# B&R Automation Studio project NAINV104C00R8L515F00 (part 15)

#### Act_OptP1081Navi.st
```iecst
ACTION Act_OptP1081Navi:

	IF tyP1081UsrMgmtUsrAccessRgt.tyNaviBack.tyBtnBack.bRtCompl = TRUE THEN
		tyP1081UsrMgmtUsrAccessRgt.tyNaviBack.tyBtnBack.bRtCompl	:= FALSE;
		tyP1081UsrMgmtUsrAccessRgt.tyNaviBack.tyBtnBack.bValue		:= FALSE;

		eChgPage	:= UIP1080UsrMgmt;
	END_IF

END_ACTION
```

#### Act_OptP1081Load.st
```iecst
ACTION Act_OptP1081Load:

	IF tyP1081UsrMgmtUsrAccessRgt.tyUsrAccessRgtSel.tyDrpDnLevel.bRtCompl = TRUE THEN
		tyP1081UsrMgmtUsrAccessRgt.tyUsrAccessRgtSel.tyDrpDnLevel.bRtCompl	:= FALSE;

		CASE tyP1081UsrMgmtUsrAccessRgt.tyUsrAccessRgtSel.tyDrpDnLevel.usiValueIdx OF
			0:
				p_tyP1081UsrMgmtUsrAccessRgt ACCESS ADR(tyP1081UsrMgmtUsrAccessRgt.tyUsrAccessRgtLvl1);
			1:
				p_tyP1081UsrMgmtUsrAccessRgt ACCESS ADR(tyP1081UsrMgmtUsrAccessRgt.tyUsrAccessRgtLvl2);
			2:
				p_tyP1081UsrMgmtUsrAccessRgt ACCESS ADR(tyP1081UsrMgmtUsrAccessRgt.tyUsrAccessRgtLvl3);
		END_CASE

	END_IF

END_ACTION
```

#### Act_OptP1081Save.st
```iecst
ACTION Act_OptP1081Save:

	//Level 1
	IF tyP1081UsrMgmtUsrAccessRgt.tyUsrAccessRgtLvl1.tyStringNm.bRtCompl 		OR tyP1081UsrMgmtUsrAccessRgt.tyUsrAccessRgtLvl1.tyBtnOps.bRtCompl
		OR tyP1081UsrMgmtUsrAccessRgt.tyUsrAccessRgtLvl1.tyBtnProdSel.bRtCompl	OR tyP1081UsrMgmtUsrAccessRgt.tyUsrAccessRgtLvl1.tyBtnMagSel.bRtCompl
		OR tyP1081UsrMgmtUsrAccessRgt.tyUsrAccessRgtLvl1.tyBtnMcInfo.bRtCompl	OR tyP1081UsrMgmtUsrAccessRgt.tyUsrAccessRgtLvl1.tyBtnAlm.bRtCompl
		OR tyP1081UsrMgmtUsrAccessRgt.tyUsrAccessRgtLvl1.tyBtnBffrInfo.bRtCompl	OR tyP1081UsrMgmtUsrAccessRgt.tyUsrAccessRgtLvl1.tyBtnOvenInfo.bRtCompl
		OR tyP1081UsrMgmtUsrAccessRgt.tyUsrAccessRgtLvl1.tyBtnMagInfo.bRtCompl	OR tyP1081UsrMgmtUsrAccessRgt.tyUsrAccessRgtLvl1.tyBtnLFCtrl.bRtCompl
		OR tyP1081UsrMgmtUsrAccessRgt.tyUsrAccessRgtLvl1.tyBtnManual.bRtCompl	OR tyP1081UsrMgmtUsrAccessRgt.tyUsrAccessRgtLvl1.tyBtnSimu.bRtCompl
		OR tyP1081UsrMgmtUsrAccessRgt.tyUsrAccessRgtLvl1.tyBtnProdSet.bRtCompl	OR tyP1081UsrMgmtUsrAccessRgt.tyUsrAccessRgtLvl1.tyBtnMagSet.bRtCompl
		OR tyP1081UsrMgmtUsrAccessRgt.tyUsrAccessRgtLvl1.tyBtnMcSet.bRtCompl	OR tyP1081UsrMgmtUsrAccessRgt.tyUsrAccessRgtLvl1.tyBtnLang.bRtCompl
		OR tyP1081UsrMgmtUsrAccessRgt.tyUsrAccessRgtLvl1.tyBtnLFSet.bRtCompl	OR tyP1081UsrMgmtUsrAccessRgt.tyUsrAccessRgtLvl1.tyBtnChgParam.bRtCompl
		OR tyP1081UsrMgmtUsrAccessRgt.tyUsrAccessRgtLvl1.tyBtnManualFBOnly.bRtCompl
		//Level 2
		OR tyP1081UsrMgmtUsrAccessRgt.tyUsrAccessRgtLvl2.tyStringNm.bRtCompl 	OR tyP1081UsrMgmtUsrAccessRgt.tyUsrAccessRgtLvl2.tyBtnOps.bRtCompl
		OR tyP1081UsrMgmtUsrAccessRgt.tyUsrAccessRgtLvl2.tyBtnProdSel.bRtCompl	OR tyP1081UsrMgmtUsrAccessRgt.tyUsrAccessRgtLvl2.tyBtnMagSel.bRtCompl
		OR tyP1081UsrMgmtUsrAccessRgt.tyUsrAccessRgtLvl2.tyBtnMcInfo.bRtCompl	OR tyP1081UsrMgmtUsrAccessRgt.tyUsrAccessRgtLvl2.tyBtnAlm.bRtCompl
		OR tyP1081UsrMgmtUsrAccessRgt.tyUsrAccessRgtLvl2.tyBtnBffrInfo.bRtCompl	OR tyP1081UsrMgmtUsrAccessRgt.tyUsrAccessRgtLvl2.tyBtnOvenInfo.bRtCompl
		OR tyP1081UsrMgmtUsrAccessRgt.tyUsrAccessRgtLvl2.tyBtnMagInfo.bRtCompl	OR tyP1081UsrMgmtUsrAccessRgt.tyUsrAccessRgtLvl2.tyBtnLFCtrl.bRtCompl
		OR tyP1081UsrMgmtUsrAccessRgt.tyUsrAccessRgtLvl2.tyBtnManual.bRtCompl	OR tyP1081UsrMgmtUsrAccessRgt.tyUsrAccessRgtLvl2.tyBtnSimu.bRtCompl
		OR tyP1081UsrMgmtUsrAccessRgt.tyUsrAccessRgtLvl2.tyBtnProdSet.bRtCompl	OR tyP1081UsrMgmtUsrAccessRgt.tyUsrAccessRgtLvl2.tyBtnMagSet.bRtCompl
		OR tyP1081UsrMgmtUsrAccessRgt.tyUsrAccessRgtLvl2.tyBtnMcSet.bRtCompl	OR tyP1081UsrMgmtUsrAccessRgt.tyUsrAccessRgtLvl2.tyBtnLang.bRtCompl
		OR tyP1081UsrMgmtUsrAccessRgt.tyUsrAccessRgtLvl2.tyBtnLFSet.bRtCompl	OR tyP1081UsrMgmtUsrAccessRgt.tyUsrAccessRgtLvl2.tyBtnChgParam.bRtCompl
		OR tyP1081UsrMgmtUsrAccessRgt.tyUsrAccessRgtLvl2.tyBtnManualFBOnly.bRtCompl

		//Level 3
		OR tyP1081UsrMgmtUsrAccessRgt.tyUsrAccessRgtLvl3.tyStringNm.bRtCompl 	OR tyP1081UsrMgmtUsrAccessRgt.tyUsrAccessRgtLvl3.tyBtnOps.bRtCompl
		OR tyP1081UsrMgmtUsrAccessRgt.tyUsrAccessRgtLvl3.tyBtnProdSel.bRtCompl	OR tyP1081UsrMgmtUsrAccessRgt.tyUsrAccessRgtLvl3.tyBtnMagSel.bRtCompl
		OR tyP1081UsrMgmtUsrAccessRgt.tyUsrAccessRgtLvl3.tyBtnMcInfo.bRtCompl	OR tyP1081UsrMgmtUsrAccessRgt.tyUsrAccessRgtLvl3.tyBtnAlm.bRtCompl
		OR tyP1081UsrMgmtUsrAccessRgt.tyUsrAccessRgtLvl3.tyBtnBffrInfo.bRtCompl	OR tyP1081UsrMgmtUsrAccessRgt.tyUsrAccessRgtLvl3.tyBtnOvenInfo.bRtCompl
		OR tyP1081UsrMgmtUsrAccessRgt.tyUsrAccessRgtLvl3.tyBtnMagInfo.bRtCompl	OR tyP1081UsrMgmtUsrAccessRgt.tyUsrAccessRgtLvl3.tyBtnLFCtrl.bRtCompl
		OR tyP1081UsrMgmtUsrAccessRgt.tyUsrAccessRgtLvl3.tyBtnManual.bRtCompl	OR tyP1081UsrMgmtUsrAccessRgt.tyUsrAccessRgtLvl3.tyBtnSimu.bRtCompl
		OR tyP1081UsrMgmtUsrAccessRgt.tyUsrAccessRgtLvl3.tyBtnProdSet.bRtCompl	OR tyP1081UsrMgmtUsrAccessRgt.tyUsrAccessRgtLvl3.tyBtnMagSet.bRtCompl
		OR tyP1081UsrMgmtUsrAccessRgt.tyUsrAccessRgtLvl3.tyBtnMcSet.bRtCompl	OR tyP1081UsrMgmtUsrAccessRgt.tyUsrAccessRgtLvl3.tyBtnLang.bRtCompl
		OR tyP1081UsrMgmtUsrAccessRgt.tyUsrAccessRgtLvl3.tyBtnLFSet.bRtCompl	OR tyP1081UsrMgmtUsrAccessRgt.tyUsrAccessRgtLvl3.tyBtnChgParam.bRtCompl
		OR tyP1081UsrMgmtUsrAccessRgt.tyUsrAccessRgtLvl3.tyBtnManualFBOnly.bRtCompl
		THEN

		fUIInRtStatHide(ADR(tyCommon.tySet.tyBtnSave.uiMaskRtStat));

		//Level 1
		tyP1081UsrMgmtUsrAccessRgt.tyUsrAccessRgtLvl1.tyStringNm.bRtCompl 		:= FALSE;
		tyP1081UsrMgmtUsrAccessRgt.tyUsrAccessRgtLvl1.tyBtnOps.bRtCompl 		:= FALSE;
		tyP1081UsrMgmtUsrAccessRgt.tyUsrAccessRgtLvl1.tyBtnProdSel.bRtCompl 	:= FALSE;
		tyP1081UsrMgmtUsrAccessRgt.tyUsrAccessRgtLvl1.tyBtnMagSel.bRtCompl 		:= FALSE;
		tyP1081UsrMgmtUsrAccessRgt.tyUsrAccessRgtLvl1.tyBtnMcInfo.bRtCompl		:= FALSE;
		tyP1081UsrMgmtUsrAccessRgt.tyUsrAccessRgtLvl1.tyBtnAlm.bRtCompl			:= FALSE;
		tyP1081UsrMgmtUsrAccessRgt.tyUsrAccessRgtLvl1.tyBtnBffrInfo.bRtCompl	:= FALSE;
		tyP1081UsrMgmtUsrAccessRgt.tyUsrAccessRgtLvl1.tyBtnOvenInfo.bRtCompl	:= FALSE;
		tyP1081UsrMgmtUsrAccessRgt.tyUsrAccessRgtLvl1.tyBtnMagInfo.bRtCompl		:= FALSE;
		tyP1081UsrMgmtUsrAccessRgt.tyUsrAccessRgtLvl1.tyBtnLFCtrl.bRtCompl		:= FALSE;
		tyP1081UsrMgmtUsrAccessRgt.tyUsrAccessRgtLvl1.tyBtnManual.bRtCompl		:= FALSE;
		tyP1081UsrMgmtUsrAccessRgt.tyUsrAccessRgtLvl1.tyBtnSimu.bRtCompl		:= FALSE;
		tyP1081UsrMgmtUsrAccessRgt.tyUsrAccessRgtLvl1.tyBtnProdSet.bRtCompl		:= FALSE;
		tyP1081UsrMgmtUsrAccessRgt.tyUsrAccessRgtLvl1.tyBtnMagSet.bRtCompl		:= FALSE;
		tyP1081UsrMgmtUsrAccessRgt.tyUsrAccessRgtLvl1.tyBtnMcSet.bRtCompl		:= FALSE;
		tyP1081UsrMgmtUsrAccessRgt.tyUsrAccessRgtLvl1.tyBtnLang.bRtCompl		:= FALSE;
		tyP1081UsrMgmtUsrAccessRgt.tyUsrAccessRgtLvl1.tyBtnLFSet.bRtCompl		:= FALSE;
		tyP1081UsrMgmtUsrAccessRgt.tyUsrAccessRgtLvl1.tyBtnChgParam.bRtCompl	:= FALSE;
		tyP1081UsrMgmtUsrAccessRgt.tyUsrAccessRgtLvl1.tyBtnManualFBOnly.bRtCompl:= FALSE;

		//Level 2
		tyP1081UsrMgmtUsrAccessRgt.tyUsrAccessRgtLvl2.tyStringNm.bRtCompl 		:= FALSE;
		tyP1081UsrMgmtUsrAccessRgt.tyUsrAccessRgtLvl2.tyBtnOps.bRtCompl 		:= FALSE;
		tyP1081UsrMgmtUsrAccessRgt.tyUsrAccessRgtLvl2.tyBtnProdSel.bRtCompl 	:= FALSE;
		tyP1081UsrMgmtUsrAccessRgt.tyUsrAccessRgtLvl2.tyBtnMagSel.bRtCompl 		:= FALSE;
		tyP1081UsrMgmtUsrAccessRgt.tyUsrAccessRgtLvl2.tyBtnMcInfo.bRtCompl		:= FALSE;
		tyP1081UsrMgmtUsrAccessRgt.tyUsrAccessRgtLvl2.tyBtnAlm.bRtCompl			:= FALSE;
		tyP1081UsrMgmtUsrAccessRgt.tyUsrAccessRgtLvl2.tyBtnBffrInfo.bRtCompl	:= FALSE;
		tyP1081UsrMgmtUsrAccessRgt.tyUsrAccessRgtLvl2.tyBtnOvenInfo.bRtCompl	:= FALSE;
		tyP1081UsrMgmtUsrAccessRgt.tyUsrAccessRgtLvl2.tyBtnMagInfo.bRtCompl		:= FALSE;
		tyP1081UsrMgmtUsrAccessRgt.tyUsrAccessRgtLvl2.tyBtnLFCtrl.bRtCompl		:= FALSE;
		tyP1081UsrMgmtUsrAccessRgt.tyUsrAccessRgtLvl2.tyBtnManual.bRtCompl		:= FALSE;
		tyP1081UsrMgmtUsrAccessRgt.tyUsrAccessRgtLvl2.tyBtnSimu.bRtCompl		:= FALSE;
		tyP1081UsrMgmtUsrAccessRgt.tyUsrAccessRgtLvl2.tyBtnProdSet.bRtCompl		:= FALSE;
		tyP1081UsrMgmtUsrAccessRgt.tyUsrAccessRgtLvl2.tyBtnMagSet.bRtCompl		:= FALSE;
		tyP1081UsrMgmtUsrAccessRgt.tyUsrAccessRgtLvl2.tyBtnMcSet.bRtCompl		:= FALSE;
		tyP1081UsrMgmtUsrAccessRgt.tyUsrAccessRgtLvl2.tyBtnLang.bRtCompl		:= FALSE;
		tyP1081UsrMgmtUsrAccessRgt.tyUsrAccessRgtLvl2.tyBtnLFSet.bRtCompl		:= FALSE;
		tyP1081UsrMgmtUsrAccessRgt.tyUsrAccessRgtLvl2.tyBtnChgParam.bRtCompl	:= FALSE;
		tyP1081UsrMgmtUsrAccessRgt.tyUsrAccessRgtLvl2.tyBtnManualFBOnly.bRtCompl:= FALSE;

		//Level 3
		tyP1081UsrMgmtUsrAccessRgt.tyUsrAccessRgtLvl3.tyStringNm.bRtCompl 		:= FALSE;
		tyP1081UsrMgmtUsrAccessRgt.tyUsrAccessRgtLvl3.tyBtnOps.bRtCompl 		:= FALSE;
		tyP1081UsrMgmtUsrAccessRgt.tyUsrAccessRgtLvl3.tyBtnProdSel.bRtCompl 	:= FALSE;
		tyP1081UsrMgmtUsrAccessRgt.tyUsrAccessRgtLvl3.tyBtnMagSel.bRtCompl 		:= FALSE;
		tyP1081UsrMgmtUsrAccessRgt.tyUsrAccessRgtLvl3.tyBtnMcInfo.bRtCompl		:= FALSE;
		tyP1081UsrMgmtUsrAccessRgt.tyUsrAccessRgtLvl3.tyBtnAlm.bRtCompl			:= FALSE;
		tyP1081UsrMgmtUsrAccessRgt.tyUsrAccessRgtLvl3.tyBtnBffrInfo.bRtCompl	:= FALSE;
		tyP1081UsrMgmtUsrAccessRgt.tyUsrAccessRgtLvl3.tyBtnOvenInfo.bRtCompl	:= FALSE;
		tyP1081UsrMgmtUsrAccessRgt.tyUsrAccessRgtLvl3.tyBtnMagInfo.bRtCompl		:= FALSE;
		tyP1081UsrMgmtUsrAccessRgt.tyUsrAccessRgtLvl3.tyBtnLFCtrl.bRtCompl		:= FALSE;
		tyP1081UsrMgmtUsrAccessRgt.tyUsrAccessRgtLvl3.tyBtnManual.bRtCompl		:= FALSE;
		tyP1081UsrMgmtUsrAccessRgt.tyUsrAccessRgtLvl3.tyBtnSimu.bRtCompl		:= FALSE;
		tyP1081UsrMgmtUsrAccessRgt.tyUsrAccessRgtLvl3.tyBtnProdSet.bRtCompl		:= FALSE;
		tyP1081UsrMgmtUsrAccessRgt.tyUsrAccessRgtLvl3.tyBtnMagSet.bRtCompl		:= FALSE;
		tyP1081UsrMgmtUsrAccessRgt.tyUsrAccessRgtLvl3.tyBtnMcSet.bRtCompl		:= FALSE;
		tyP1081UsrMgmtUsrAccessRgt.tyUsrAccessRgtLvl3.tyBtnLang.bRtCompl		:= FALSE;
		tyP1081UsrMgmtUsrAccessRgt.tyUsrAccessRgtLvl3.tyBtnLFSet.bRtCompl		:= FALSE;
		tyP1081UsrMgmtUsrAccessRgt.tyUsrAccessRgtLvl3.tyBtnChgParam.bRtCompl	:= FALSE;
		tyP1081UsrMgmtUsrAccessRgt.tyUsrAccessRgtLvl3.tyBtnManualFBOnly.bRtCompl:= FALSE;

	END_IF

	IF tyCommon.tySet.tyBtnSave.bRtCompl = TRUE THEN
		//Save Param
		CASE tyP1081UsrMgmtUsrAccessRgt.tyUsrAccessRgtSel.tyDrpDnLevel.usiValueIdx OF
			0:
				tyUsrMgmtAccessRightLvl1Wr.sNm			:= tyP1081UsrMgmtUsrAccessRgt.tyUsrAccessRgtLvl1.tyStringNm.sValue;
				tyUsrMgmtAccessRightLvl1Wr.bOpt			:= tyP1081UsrMgmtUsrAccessRgt.tyUsrAccessRgtLvl1.tyBtnOps.bValue;
				tyUsrMgmtAccessRightLvl1Wr.bProdSel		:= tyP1081UsrMgmtUsrAccessRgt.tyUsrAccessRgtLvl1.tyBtnProdSel.bValue;
				tyUsrMgmtAccessRightLvl1Wr.bMagSel		:= tyP1081UsrMgmtUsrAccessRgt.tyUsrAccessRgtLvl1.tyBtnMagSel.bValue;
				tyUsrMgmtAccessRightLvl1Wr.bMcInfo		:= tyP1081UsrMgmtUsrAccessRgt.tyUsrAccessRgtLvl1.tyBtnMcInfo.bValue;
				tyUsrMgmtAccessRightLvl1Wr.bAlm			:= tyP1081UsrMgmtUsrAccessRgt.tyUsrAccessRgtLvl1.tyBtnAlm.bValue;
				tyUsrMgmtAccessRightLvl1Wr.bBffrInfo	:= tyP1081UsrMgmtUsrAccessRgt.tyUsrAccessRgtLvl1.tyBtnBffrInfo.bValue;
				tyUsrMgmtAccessRightLvl1Wr.bOvenInfo	:= tyP1081UsrMgmtUsrAccessRgt.tyUsrAccessRgtLvl1.tyBtnOvenInfo.bValue;
				tyUsrMgmtAccessRightLvl1Wr.bMagInfo		:= tyP1081UsrMgmtUsrAccessRgt.tyUsrAccessRgtLvl1.tyBtnMagInfo.bValue;
				tyUsrMgmtAccessRightLvl1Wr.bLFCtrl		:= tyP1081UsrMgmtUsrAccessRgt.tyUsrAccessRgtLvl1.tyBtnLFCtrl.bValue;
				tyUsrMgmtAccessRightLvl1Wr.bManual		:= tyP1081UsrMgmtUsrAccessRgt.tyUsrAccessRgtLvl1.tyBtnManual.bValue;
				tyUsrMgmtAccessRightLvl1Wr.bSimulation	:= tyP1081UsrMgmtUsrAccessRgt.tyUsrAccessRgtLvl1.tyBtnSimu.bValue;
				tyUsrMgmtAccessRightLvl1Wr.bProdSet		:= tyP1081UsrMgmtUsrAccessRgt.tyUsrAccessRgtLvl1.tyBtnProdSet.bValue;
				tyUsrMgmtAccessRightLvl1Wr.bMagSet		:= tyP1081UsrMgmtUsrAccessRgt.tyUsrAccessRgtLvl1.tyBtnMagSet.bValue;
				tyUsrMgmtAccessRightLvl1Wr.bMcSet		:= tyP1081UsrMgmtUsrAccessRgt.tyUsrAccessRgtLvl1.tyBtnMcSet.bValue;
				tyUsrMgmtAccessRightLvl1Wr.bLang		:= tyP1081UsrMgmtUsrAccessRgt.tyUsrAccessRgtLvl1.tyBtnLang.bValue;
				tyUsrMgmtAccessRightLvl1Wr.bLFSet		:= tyP1081UsrMgmtUsrAccessRgt.tyUsrAccessRgtLvl1.tyBtnLFSet.bValue;
				tyUsrMgmtAccessRightLvl1Wr.bChgParam	:= tyP1081UsrMgmtUsrAccessRgt.tyUsrAccessRgtLvl1.tyBtnChgParam.bValue;
				tyUsrMgmtAccessRightLvl1Wr.bManualFBOnly:= tyP1081UsrMgmtUsrAccessRgt.tyUsrAccessRgtLvl1.tyBtnManualFBOnly.bValue;

			1:
				tyUsrMgmtAccessRightLvl2Wr.sNm			:= tyP1081UsrMgmtUsrAccessRgt.tyUsrAccessRgtLvl2.tyStringNm.sValue;
				tyUsrMgmtAccessRightLvl2Wr.bOpt			:= tyP1081UsrMgmtUsrAccessRgt.tyUsrAccessRgtLvl2.tyBtnOps.bValue;
				tyUsrMgmtAccessRightLvl2Wr.bProdSel		:= tyP1081UsrMgmtUsrAccessRgt.tyUsrAccessRgtLvl2.tyBtnProdSel.bValue;
				tyUsrMgmtAccessRightLvl2Wr.bMagSel		:= tyP1081UsrMgmtUsrAccessRgt.tyUsrAccessRgtLvl2.tyBtnMagSel.bValue;
				tyUsrMgmtAccessRightLvl2Wr.bMcInfo		:= tyP1081UsrMgmtUsrAccessRgt.tyUsrAccessRgtLvl2.tyBtnMcInfo.bValue;
				tyUsrMgmtAccessRightLvl2Wr.bAlm			:= tyP1081UsrMgmtUsrAccessRgt.tyUsrAccessRgtLvl2.tyBtnAlm.bValue;
				tyUsrMgmtAccessRightLvl2Wr.bBffrInfo	:= tyP1081UsrMgmtUsrAccessRgt.tyUsrAccessRgtLvl2.tyBtnBffrInfo.bValue;
				tyUsrMgmtAccessRightLvl2Wr.bOvenInfo	:= tyP1081UsrMgmtUsrAccessRgt.tyUsrAccessRgtLvl2.tyBtnOvenInfo.bValue;
				tyUsrMgmtAccessRightLvl2Wr.bMagInfo		:= tyP1081UsrMgmtUsrAccessRgt.tyUsrAccessRgtLvl2.tyBtnMagInfo.bValue;
				tyUsrMgmtAccessRightLvl2Wr.bLFCtrl		:= tyP1081UsrMgmtUsrAccessRgt.tyUsrAccessRgtLvl2.tyBtnLFCtrl.bValue;
				tyUsrMgmtAccessRightLvl2Wr.bManual		:= tyP1081UsrMgmtUsrAccessRgt.tyUsrAccessRgtLvl2.tyBtnManual.bValue;
				tyUsrMgmtAccessRightLvl2Wr.bSimulation	:= tyP1081UsrMgmtUsrAccessRgt.tyUsrAccessRgtLvl2.tyBtnSimu.bValue;
				tyUsrMgmtAccessRightLvl2Wr.bProdSet		:= tyP1081UsrMgmtUsrAccessRgt.tyUsrAccessRgtLvl2.tyBtnProdSet.bValue;
				tyUsrMgmtAccessRightLvl2Wr.bMagSet		:= tyP1081UsrMgmtUsrAccessRgt.tyUsrAccessRgtLvl2.tyBtnMagSet.bValue;
				tyUsrMgmtAccessRightLvl2Wr.bMcSet		:= tyP1081UsrMgmtUsrAccessRgt.tyUsrAccessRgtLvl2.tyBtnMcSet.bValue;
				tyUsrMgmtAccessRightLvl2Wr.bLang		:= tyP1081UsrMgmtUsrAccessRgt.tyUsrAccessRgtLvl2.tyBtnLang.bValue;
				tyUsrMgmtAccessRightLvl2Wr.bLFSet		:= tyP1081UsrMgmtUsrAccessRgt.tyUsrAccessRgtLvl2.tyBtnLFSet.bValue;
				tyUsrMgmtAccessRightLvl2Wr.bChgParam	:= tyP1081UsrMgmtUsrAccessRgt.tyUsrAccessRgtLvl2.tyBtnChgParam.bValue;
				tyUsrMgmtAccessRightLvl2Wr.bManualFBOnly:= tyP1081UsrMgmtUsrAccessRgt.tyUsrAccessRgtLvl2.tyBtnManualFBOnly.bValue;

			2:
				tyUsrMgmtAccessRightLvl3Wr.sNm			:= tyP1081UsrMgmtUsrAccessRgt.tyUsrAccessRgtLvl3.tyStringNm.sValue;
				tyUsrMgmtAccessRightLvl3Wr.bOpt			:= tyP1081UsrMgmtUsrAccessRgt.tyUsrAccessRgtLvl3.tyBtnOps.bValue;
				tyUsrMgmtAccessRightLvl3Wr.bProdSel		:= tyP1081UsrMgmtUsrAccessRgt.tyUsrAccessRgtLvl3.tyBtnProdSel.bValue;
				tyUsrMgmtAccessRightLvl3Wr.bMagSel		:= tyP1081UsrMgmtUsrAccessRgt.tyUsrAccessRgtLvl3.tyBtnMagSel.bValue;
				tyUsrMgmtAccessRightLvl3Wr.bMcInfo		:= tyP1081UsrMgmtUsrAccessRgt.tyUsrAccessRgtLvl3.tyBtnMcInfo.bValue;
				tyUsrMgmtAccessRightLvl3Wr.bAlm			:= tyP1081UsrMgmtUsrAccessRgt.tyUsrAccessRgtLvl3.tyBtnAlm.bValue;
				tyUsrMgmtAccessRightLvl3Wr.bBffrInfo	:= tyP1081UsrMgmtUsrAccessRgt.tyUsrAccessRgtLvl3.tyBtnBffrInfo.bValue;
				tyUsrMgmtAccessRightLvl3Wr.bOvenInfo	:= tyP1081UsrMgmtUsrAccessRgt.tyUsrAccessRgtLvl3.tyBtnOvenInfo.bValue;
				tyUsrMgmtAccessRightLvl3Wr.bMagInfo		:= tyP1081UsrMgmtUsrAccessRgt.tyUsrAccessRgtLvl3.tyBtnMagInfo.bValue;
				tyUsrMgmtAccessRightLvl3Wr.bLFCtrl		:= tyP1081UsrMgmtUsrAccessRgt.tyUsrAccessRgtLvl3.tyBtnLFCtrl.bValue;
				tyUsrMgmtAccessRightLvl3Wr.bManual		:= tyP1081UsrMgmtUsrAccessRgt.tyUsrAccessRgtLvl3.tyBtnManual.bValue;
				tyUsrMgmtAccessRightLvl3Wr.bSimulation	:= tyP1081UsrMgmtUsrAccessRgt.tyUsrAccessRgtLvl3.tyBtnSimu.bValue;
				tyUsrMgmtAccessRightLvl3Wr.bProdSet		:= tyP1081UsrMgmtUsrAccessRgt.tyUsrAccessRgtLvl3.tyBtnProdSet.bValue;
				tyUsrMgmtAccessRightLvl3Wr.bMagSet		:= tyP1081UsrMgmtUsrAccessRgt.tyUsrAccessRgtLvl3.tyBtnMagSet.bValue;
				tyUsrMgmtAccessRightLvl3Wr.bMcSet		:= tyP1081UsrMgmtUsrAccessRgt.tyUsrAccessRgtLvl3.tyBtnMcSet.bValue;
				tyUsrMgmtAccessRightLvl3Wr.bLang		:= tyP1081UsrMgmtUsrAccessRgt.tyUsrAccessRgtLvl3.tyBtnLang.bValue;
				tyUsrMgmtAccessRightLvl3Wr.bLFSet		:= tyP1081UsrMgmtUsrAccessRgt.tyUsrAccessRgtLvl3.tyBtnLFSet.bValue;
				tyUsrMgmtAccessRightLvl3Wr.bChgParam	:= tyP1081UsrMgmtUsrAccessRgt.tyUsrAccessRgtLvl3.tyBtnChgParam.bValue;
				tyUsrMgmtAccessRightLvl3Wr.bManualFBOnly:= tyP1081UsrMgmtUsrAccessRgt.tyUsrAccessRgtLvl3.tyBtnManualFBOnly.bValue;

		END_CASE

		eUsrMgmtAct	:= UsrMgmtActSaveAccessRight;

		IF p_eUsrMgmtStat = UsrMgmtActSaveAccessRight AND p_eUsrMgmtStatus = Done THEN
			eUsrMgmtAct	:= UsrMgmtActIdle;

			//Backup Param
			tyP1081UsrMgmtUsrAccessRgt.tyUsrAccessRgtLvl1BkUp	:= tyP1081UsrMgmtUsrAccessRgt.tyUsrAccessRgtLvl1;
			tyP1081UsrMgmtUsrAccessRgt.tyUsrAccessRgtLvl2BkUp	:= tyP1081UsrMgmtUsrAccessRgt.tyUsrAccessRgtLvl2;
			tyP1081UsrMgmtUsrAccessRgt.tyUsrAccessRgtLvl3BkUp	:= tyP1081UsrMgmtUsrAccessRgt.tyUsrAccessRgtLvl3;

			CASE tyP1081UsrMgmtUsrAccessRgt.tyUsrAccessRgtSel.tyDrpDnLevel.usiValueIdx OF
				0:
					tyProperty.tyUITxtSnippets.sUsrMgmtUsrLv1Nm	:= tyP1081UsrMgmtUsrAccessRgt.tyUsrAccessRgtLvl1.tyStringNm.sValue;
				1:
					tyProperty.tyUITxtSnippets.sUsrMgmtUsrLv2Nm	:= tyP1081UsrMgmtUsrAccessRgt.tyUsrAccessRgtLvl2.tyStringNm.sValue;
				2:
					tyProperty.tyUITxtSnippets.sUsrMgmtUsrLv3Nm	:= tyP1081UsrMgmtUsrAccessRgt.tyUsrAccessRgtLvl3.tyStringNm.sValue;
			END_CASE

			tyCommon.tySet.tyBtnSave.bRtCompl	:= FALSE;

			fUIInRtStatOff(ADR(tyCommon.tySet.tyBtnSave.uiMaskRtStat));

		ELSIF p_eUsrMgmtStatus = Error THEN
			p_tyC0008MsgBox ACCESS ADR(tyP1081UsrMgmtUsrAccessRgt.tyMsgBoxSaveErr);

			IF tyP1081UsrMgmtUsrAccessRgt.tyMsgBoxSaveErr.tyBtnNo.bRtCompl = TRUE THEN
				tyP1081UsrMgmtUsrAccessRgt.tyMsgBoxSaveErr.tyBtnNo.bRtCompl	:= FALSE;
				tyP1081UsrMgmtUsrAccessRgt.tyMsgBoxSaveErr.tyBtnNo.bValue	:= FALSE;

				p_tyC0008MsgBox ACCESS ADR(tyP1081UsrMgmtUsrAccessRgt.tyMsgBoxHide);

				//Recover Param
				tyUsrMgmtAccessRightLvl1Wr	:= p_tyUsrMgmtFullData.tyAccessRightLvl1;
				tyUsrMgmtAccessRightLvl2Wr	:= p_tyUsrMgmtFullData.tyAccessRightLvl2;
				tyUsrMgmtAccessRightLvl3Wr	:= p_tyUsrMgmtFullData.tyAccessRightLvl3;

				tyP1081UsrMgmtUsrAccessRgt.tyUsrAccessRgtLvl1	:= tyP1081UsrMgmtUsrAccessRgt.tyUsrAccessRgtLvl1BkUp;
				tyP1081UsrMgmtUsrAccessRgt.tyUsrAccessRgtLvl2	:= tyP1081UsrMgmtUsrAccessRgt.tyUsrAccessRgtLvl2BkUp;
				tyP1081UsrMgmtUsrAccessRgt.tyUsrAccessRgtLvl3	:= tyP1081UsrMgmtUsrAccessRgt.tyUsrAccessRgtLvl3BkUp;

				tyCommon.tySet.tyBtnSave.bRtCompl	:= FALSE;

				fUIInRtStatOff(ADR(tyCommon.tySet.tyBtnSave.uiMaskRtStat));

			END_IF

		END_IF

	END_IF

END_ACTION
```

#### Act_OptP1081Keypad.st
```iecst
ACTION Act_OptP1081Keypad:

	IF fUIOutRtStatTPIsOpen(ADR(tyP1081UsrMgmtUsrAccessRgt.tyUsrAccessRgtLvl1.tyStringNm.uiRtStat)) = TRUE THEN
		tyProperty.tyKeypad.tyTxtTitle.sTxt	:= tyP1081UsrMgmtUsrAccessRgt.tyUsrAccessRgtLvl1.tyStringNm.sKeypadTitle;

	ELSIF fUIOutRtStatTPIsOpen(ADR(tyP1081UsrMgmtUsrAccessRgt.tyUsrAccessRgtLvl2.tyStringNm.uiRtStat)) = TRUE THEN
		tyProperty.tyKeypad.tyTxtTitle.sTxt	:= tyP1081UsrMgmtUsrAccessRgt.tyUsrAccessRgtLvl2.tyStringNm.sKeypadTitle;

	ELSIF fUIOutRtStatTPIsOpen(ADR(tyP1081UsrMgmtUsrAccessRgt.tyUsrAccessRgtLvl3.tyStringNm.uiRtStat)) = TRUE THEN
		tyProperty.tyKeypad.tyTxtTitle.sTxt	:= tyP1081UsrMgmtUsrAccessRgt.tyUsrAccessRgtLvl3.tyStringNm.sKeypadTitle;

	END_IF

END_ACTION
```

#### Act_OptP0002ToP1081UnlockCoverPB.st
```iecst
ACTION Act_OptP0002ToP1081UnlockCoverPB:

	IF p_tyNtParamCurr.tyDOSettings.diBypassTopCover1 > 0 THEN

		IF p_bAlarmErr THEN
			bCoverPB1Timer := FALSE;
			fbCoverPB1CountDownTm( IN := FALSE);
			tyP0200OpsGen.tyOps.tyBtnBypassTopCover1.bValue 	:=FALSE;
			tyP0201OpsConv.tyOps.tyBtnBypassTopCover1.bValue	:=FALSE;
		END_IF

		//Physical Unlock Cover Button 1
		IF EDGENEG(p_tyDI.bCoverUnlockPB1) THEN
			IF p_tyDI.bCoverSWSig2 = TRUE THEN
				IF tyP0200OpsGen.tyOps.tyBtnBypassTopCover1.bValue = FALSE THEN
					tyP0200OpsGen.tyOps.tyBtnBypassTopCover1.bValue 	:= TRUE;
					tyP0201OpsConv.tyOps.tyBtnBypassTopCover1.bValue	:= tyP0200OpsGen.tyOps.tyBtnBypassTopCover1.bValue;
					bCoverPB1Timer := TRUE;
				ELSE
					tyP0200OpsGen.tyOps.tyBtnBypassTopCover1.bValue 	:= FALSE;
					tyP0201OpsConv.tyOps.tyBtnBypassTopCover1.bValue	:= tyP0200OpsGen.tyOps.tyBtnBypassTopCover1.bValue;
					bCoverPB1Timer := FALSE;
				END_IF
			END_IF
		END_IF

		//Control
		IF tyP0200OpsGen.tyOps.tyBtnBypassTopCover1.bRtCompl = TRUE THEN //ok
			tyP0200OpsGen.tyOps.tyBtnBypassTopCover1.bRtCompl	:= FALSE;
			IF p_tyDI.bCoverSWSig2 = TRUE THEN
				tyP0201OpsConv.tyOps.tyBtnBypassTopCover1.bValue	:= tyP0200OpsGen.tyOps.tyBtnBypassTopCover1.bValue;
				IF tyP0200OpsGen.tyOps.tyBtnBypassTopCover1.bValue = TRUE THEN
					bCoverPB1Timer := TRUE;
				ELSE
					bCoverPB1Timer := FALSE;
				END_IF
			ELSE
				tyP0200OpsGen.tyOps.tyBtnBypassTopCover1.bValue 	:= TRUE;
				tyP0201OpsConv.tyOps.tyBtnBypassTopCover1.bValue	:= tyP0200OpsGen.tyOps.tyBtnBypassTopCover1.bValue;
			END_IF

		ELSIF tyP0201OpsConv.tyOps.tyBtnBypassTopCover1.bRtCompl = TRUE THEN //ok
			tyP0201OpsConv.tyOps.tyBtnBypassTopCover1.bRtCompl	:= FALSE;
			IF p_tyDI.bCoverSWSig = TRUE THEN
				tyP0200OpsGen.tyOps.tyBtnBypassTopCover1.bValue	:= tyP0201OpsConv.tyOps.tyBtnBypassTopCover1.bValue;
				IF tyP0201OpsConv.tyOps.tyBtnBypassTopCover1.bValue = TRUE THEN
					bCoverPB1Timer := TRUE;
				ELSE
					bCoverPB1Timer := FALSE;
				END_IF
			ELSE
				tyP0201OpsConv.tyOps.tyBtnBypassTopCover1.bValue 	:= TRUE;
				tyP0200OpsGen.tyOps.tyBtnBypassTopCover1.bValue		:= tyP0201OpsConv.tyOps.tyBtnBypassTopCover1.bValue;
			END_IF

		END_IF

		bBypassTopCover1	:= ( tyP0200OpsGen.tyOps.tyBtnBypassTopCover1.bValue) OR ( tyP0201OpsConv.tyOps.tyBtnBypassTopCover1.bValue);

		//Condition Allow
		IF (tyP0201OpsConv.tyOps.tyBtnBypassTopCover1.bValue = TRUE) THEN

			IF p_tyNtParamCurr.tyDISettings.diSafetySigFromUS > 0 THEN
				bUnlockCover1Req	:= TRUE;

				IF (p_bOpsInvertStepAWMove = FALSE) AND (p_eConvStatus <> Busy AND p_eInvertStatus <> Busy )AND
					(( p_tyDI.bInShutterCloseRS AND p_tyDI.bOutShutterCloseRS AND p_bOpsSafeMode) OR p_bOpsRun=FALSE) AND (p_tyDI.bSafetySigFromUS AND p_tyDI.bSafetySigFromDS )  THEN

					bTopCoverSwitchCoil1	:= FALSE;
				ELSE
					bTopCoverSwitchCoil1	:= TRUE;
				END_IF

			ELSE
				IF (p_bOpsInvertStepAWMove = FALSE) AND (p_eConvStatus <> Busy AND p_eInvertStatus <> Busy )AND
					((p_tyDI.bInShutterCloseRS AND p_tyDI.bOutShutterCloseRS AND p_bOpsSafeMode) OR p_bOpsRun=FALSE) THEN

					bTopCoverSwitchCoil1	:= FALSE;
				ELSE
					bTopCoverSwitchCoil1	:= TRUE;
				END_IF

			END_IF

		ELSE
			bTopCoverSwitchCoil1	:= TRUE;
			IF p_tyNtParamCurr.tyDISettings.diSafetySigFromUS > 0 THEN
				bUnlockCover1Req	:= FALSE;
				//bTopCvrUnlckToDS	:= FALSE;
			END_IF

		END_IF

		//Button Appearance
		IF bCoverPBLED1 THEN //bTopCoverSwitchCoil1 = FALSE AND tyP0200OpsGen.tyOps.tyBtnBypassTopCover1.bValue = TRUE THEN
			tyP0201OpsConv.tyOps.tyBitmapBypassTopCover1.usiValueIdx	:= 0;
			tyP0200OpsGen.tyOps.tyBitmapBypassTopCover1.usiValueIdx		:= 0;
		ELSE
			tyP0201OpsConv.tyOps.tyBitmapBypassTopCover1.usiValueIdx	:= 2;
			tyP0200OpsGen.tyOps.tyBitmapBypassTopCover1.usiValueIdx		:= 2;
		END_IF

	END_IF

	//lED 1&2

	// LED 1 & 2
	IF bTopCoverSwitchCoil1 = FALSE AND tyP0200OpsGen.tyOps.tyBtnBypassTopCover1.bValue = TRUE THEN
		bCoverPBLED1 := TRUE;
		fbCoverPBLED1BlinkTm(IN := FALSE);
	ELSIF bTopCoverSwitchCoil1 = TRUE AND tyP0200OpsGen.tyOps.tyBtnBypassTopCover1.bValue = TRUE THEN
		fbCoverPBLED1BlinkTm(IN := TRUE);
		IF fbCoverPBLED1BlinkTm.Q = TRUE THEN
			fbCoverPBLED1BlinkTm(IN := FALSE);
			IF bCoverPBLED1 = FALSE THEN
				bCoverPBLED1 := TRUE;
			ELSE
				bCoverPBLED1 := FALSE;
			END_IF
		END_IF
	ELSE
		bCoverPBLED1 := FALSE;
		fbCoverPBLED1BlinkTm(IN := FALSE);
	END_IF

	//5 Sec Time Out Cover PB1
	IF bTopCoverSwitchCoil1 = FALSE AND tyP0200OpsGen.tyOps.tyBtnBypassTopCover1.bValue = TRUE  OR bCoverPB1Timer = FALSE THEN //tyP0200OpsGen.tyOps.tyBitmapBypassTopCover1.usiValueIdx	= 1 OR bCoverPB1Timer = FALSE THEN
		fbCoverPB1CountDownTm(IN := bCoverPB1Timer);																//
		IF p_tyDI.bCoverSWSig2 = FALSE THEN
			bCoverPB1Timer := FALSE;																				//
		END_IF																										//
		//
		IF fbCoverPB1CountDownTm.Q = TRUE THEN																		//
			fbCoverPB1CountDownTm(IN := FALSE);																		//
			bCoverPB1Timer := FALSE;																				//
			tyP0200OpsGen.tyOps.tyBtnBypassTopCover1.bValue 	:= FALSE;											//
			tyP0201OpsConv.tyOps.tyBtnBypassTopCover1.bValue	:= tyP0200OpsGen.tyOps.tyBtnBypassTopCover1.bValue;	//
		END_IF																										//
	END_IF																											//

	//Lock After Close Cover
	IF EDGEPOS(p_tyDI.bCoverSWSig2) THEN																			//
		tyP0200OpsGen.tyOps.tyBtnBypassTopCover1.bValue 	:= FALSE;											//
		tyP0201OpsConv.tyOps.tyBtnBypassTopCover1.bValue	:= tyP0200OpsGen.tyOps.tyBtnBypassTopCover1.bValue;	//
	END_IF																										//

	////////////////////////////////////Machine Safety Signal To DS

	IF (p_tyDI.bUnlockCoverSigFromDS) AND (p_bOpsInvertStepAWMove = FALSE) AND
		(p_bOpsDSStandby OR ( p_eConvStatus <> Busy) AND ( p_eInvertStatus<>Busy OR p_bOutShutterExtended)) THEN

		bMachineSafetySigToDS := TRUE;
	ELSE
		bMachineSafetySigToDS := FALSE;
	END_IF

	////////////////////////////////////Machine Safety Signal To US
	IF  (p_tyDI.bUnlockCoverSigFromUS) AND  (p_bOpsInvertStepAWMove = FALSE) AND (p_bOpsUSStandby  OR ( p_eConvStatus <> Busy) AND ( p_eInvertStatus<>Busy OR p_bInShutterExtended)) THEN

		bMachineSafetySigToUS := TRUE;
	ELSE
		bMachineSafetySigToUS := FALSE;
	END_IF

END_ACTION
```

#### InputRef.var - Change By Project
```iecst
(*2020-10-08*)
(**)
(*Configuration*)
VAR
	p_eAct : REFERENCE TO eUIAction;
END_VAR
(**)
VAR
	p_bStartupRun : REFERENCE TO BOOL;
	p_eStartupStat : REFERENCE TO eStartupAction;
	p_eStartupStatus : REFERENCE TO eFBStatus;
	p_sStartupStatTxt : REFERENCE TO STRING[200];
	p_eStartupStep : REFERENCE TO eStartupStep;
	p_sStartupStepTxt : REFERENCE TO STRING[80];
	p_bStartupGetConfigDone : REFERENCE TO BOOL;
	p_bStartupMismatchSetConfigDone : REFERENCE TO BOOL;
	p_bStartupUISettingsLoadDone : REFERENCE TO BOOL;
END_VAR
(**)
VAR
	p_eTLBuzStat : REFERENCE TO eTLBuzAction;
	p_eTLBuzStatus : REFERENCE TO eFBStatus;
	p_sTLBuzStatTxt : REFERENCE TO STRING[80];
END_VAR
(**)
VAR
	p_tyAlarmCurrList : REFERENCE TO ARRAY[1..c_udiAlarmCurrMax] OF tyAlarmCurr;
	p_tyAlarmRcyList : REFERENCE TO ARRAY[1..c_udiAlarmCurrMax] OF UDINT;
	p_tyAlarmHistoryList : REFERENCE TO ARRAY[1..c_udiAlarmHistoryMax] OF STRING[200];
	p_bAlarmWarning : REFERENCE TO BOOL;
	p_bAlarmErr : REFERENCE TO BOOL;
	p_bAlarmInfo : REFERENCE TO BOOL;
	p_bAlarmInfoLF : REFERENCE TO BOOL;
	p_sAlarmInfoMsg : REFERENCE TO STRING[200];
END_VAR
(**)
VAR
	p_eRstErrStat : REFERENCE TO eRstErrAction;
	p_eRstErrStatus : REFERENCE TO eFBStatus;
	p_sRstErrStatTxt : REFERENCE TO STRING[200];
END_VAR
(**)
VAR
	p_eHWInfoStat : REFERENCE TO eHWInfoAction;
	p_eHWInfoStatus : REFERENCE TO eFBStatus;
	p_sHWInfoStatTxt : REFERENCE TO STRING[200];
	p_sHWInfoIPAddr : REFERENCE TO STRING[15];
	p_sHWInfoSubnetMask : REFERENCE TO STRING[15];
	p_udiHWInfoEthMode : REFERENCE TO UDINT;
END_VAR
(**)
VAR
	p_eProdRcpStat : REFERENCE TO eProdRcpAction;
	p_eProdRcpStatus : REFERENCE TO eFBStatus;
	p_sProdRcpStatTxt : REFERENCE TO STRING[200];
	p_tyProdRcpFilterList : REFERENCE TO ARRAY[1..c_udiProdRcpMax] OF tyProdRcpParam;
	p_tyProdRcpSortedList : REFERENCE TO ARRAY[1..c_udiProdRcpMax] OF tyProdRcpParam;
	p_tyProdRcpCurrList : REFERENCE TO ARRAY[1..c_udiProdRcpMax] OF tyProdRcpParam;
	p_tyProdRcpInfoOut : REFERENCE TO tyProdRcpParam;
	p_tyProdRcpCurrRcp0 : REFERENCE TO tyProdRcpParam;
	p_tyProdRcpCurrRcp1 : REFERENCE TO tyProdRcpParam;
	p_tyProdRcpCurrRcp2 : REFERENCE TO tyProdRcpParam;
	p_bProdRcpNmEmpty : REFERENCE TO BOOL;
	p_bProdRcpListFull : REFERENCE TO BOOL;
	p_bProdRcpNmNotExist : REFERENCE TO BOOL;
END_VAR
(**)
VAR
	p_eMpProdRcpStat : REFERENCE TO eMpProdRcpAction;
	p_eMpProdRcpStatus : REFERENCE TO eFBStatus;
END_VAR
(**)
VAR
	p_eMcParamStat : REFERENCE TO eMcParamAction;
	p_eMcParamStatus : REFERENCE TO eFBStatus;
	p_sMcParamStatTxt : REFERENCE TO STRING[200];
	p_tyMcParamCurr : REFERENCE TO tyMcParam;
END_VAR
(**)
VAR
	p_tyNtParamCurr : REFERENCE TO tyNtParam;
END_VAR
(**)
VAR
	p_eUsrMgmtStat : REFERENCE TO eUsrMgmtAction;
	p_eUsrMgmtStatus : REFERENCE TO eFBStatus;
	p_sUsrMgmtStatTxt : REFERENCE TO STRING[200];
	p_tyUsrMgmtCurrUsr : REFERENCE TO tyUsrMgmtParam;
	p_tyUsrMgmtCurrAccessRgt : REFERENCE TO tyUsrMgmtAccessRight;
	p_tyUsrMgmtAllList : REFERENCE TO ARRAY[1..c_udiUsrMgmtMax] OF tyUsrMgmtParam;
	p_tyUsrMgmtLv2List : REFERENCE TO ARRAY[1..c_udiUsrMgmtMax] OF tyUsrMgmtParam;
	p_tyUsrMgmtLv3List : REFERENCE TO ARRAY[1..c_udiUsrMgmtMax] OF tyUsrMgmtParam;
	p_tyUsrMgmtAdminList : REFERENCE TO ARRAY[1..c_udiUsrMgmtMax] OF tyUsrMgmtParam;
	p_bUsrMgmtNmEmpty : REFERENCE TO BOOL;
	p_bUsrMgmtListFull : REFERENCE TO BOOL;
	p_bUsrMgmtNmExist : REFERENCE TO BOOL;
	p_bUsrMgmtNmNotExist : REFERENCE TO BOOL;
	p_bUsrMgmtLastAdmin : REFERENCE TO BOOL;
	p_bUsrMgmtLoginSuccess : REFERENCE TO BOOL;
	p_bUsrMgmtPwMismatch : REFERENCE TO BOOL;
	p_bUsrMgmtUnableDelete : REFERENCE TO BOOL;
	p_tyUsrMgmtFullData : REFERENCE TO tyUsrMgmtFullDat;
END_VAR
(**)
VAR
	p_eUSSMEMAStat : REFERENCE TO eSMEMAAction;
	p_eUSSMEMAStatus : REFERENCE TO eFBStatus;
	p_sUSSMEMAStatTxt : REFERENCE TO STRING[80];
	p_bUSSMEMAUSRdy : REFERENCE TO BOOL;
	p_bUSSMEMAUSGdBrdRdy : REFERENCE TO BOOL;
	p_bUSSMEMADSRdy : REFERENCE TO BOOL;
	p_bUSSMEMAUSB : REFERENCE TO BOOL;
END_VAR
(**)
VAR
	p_eDSSMEMAStat : REFERENCE TO eSMEMAAction;
	p_eDSSMEMAStatus : REFERENCE TO eFBStatus;
	p_sDSSMEMAStatTxt : REFERENCE TO STRING[80];
	p_bDSSMEMAUSRdy : REFERENCE TO BOOL;
	p_bDSSMEMAUSGdBrdRdy : REFERENCE TO BOOL;
	p_bDSSMEMADSRdy : REFERENCE TO BOOL;
	p_bDSSMEMADBA : REFERENCE TO BOOL;
	p_bDSSMEMADBAStat : REFERENCE TO BOOL;
END_VAR
(**)
VAR
	p_eUSSMEMA2Stat : REFERENCE TO eSMEMAAction;
	p_eUSSMEMA2Status : REFERENCE TO eFBStatus;
	p_sUSSMEMA2StatTxt : REFERENCE TO STRING[80];
	p_bUSSMEMA2USRdy : REFERENCE TO BOOL;
	p_bUSSMEMA2USGdBrdRdy : REFERENCE TO BOOL;
	p_bUSSMEMA2DSRdy : REFERENCE TO BOOL;
	p_bUSSMEMA2USB : REFERENCE TO BOOL;
	p_bUSSMEMA2Transporting : REFERENCE TO BOOL;
END_VAR
(**)
VAR
	p_bUSHermesUSRdy : REFERENCE TO BOOL;
	p_bUSHermesDSRdy : REFERENCE TO BOOL;
	p_bUSHermesUSGdRdy : REFERENCE TO BOOL;
	p_bUSHermesDSGdRdy : REFERENCE TO BOOL;
	p_bUSHermesConnected : REFERENCE TO BOOL;
	p_bUSHermesAccDataMnl : REFERENCE TO BOOL;
END_VAR
(**)
VAR
	p_bDSHermesUSRdy : REFERENCE TO BOOL;
	p_bDSHermesDSRdy : REFERENCE TO BOOL;
	p_bDSHermesUSGdRdy : REFERENCE TO BOOL;
	p_bDSHermesDSGdRdy : REFERENCE TO BOOL;
	p_bDSHermesConnected : REFERENCE TO BOOL;
END_VAR
(**)
VAR
	p_eConvStat : REFERENCE TO eConvAction;
	p_eConvStatus : REFERENCE TO eFBStatus;
	p_sConvStatTxt : REFERENCE TO STRING[80];
	p_bConvHvBrd : REFERENCE TO BOOL;
	p_bConvGdBrd : REFERENCE TO BOOL;
END_VAR
(**)
VAR
	p_eAWOpenStat : REFERENCE TO eAWAction;
	p_eAWOpenStatus : REFERENCE TO eFBStatus;
	p_sAWOpenStatTxt : REFERENCE TO STRING[200];
	p_udiAWOpenAxisErrID : REFERENCE TO UDINT;
	p_bAWOpenAxisErr : REFERENCE TO BOOL;
	p_bAWOpenPwrOn : REFERENCE TO BOOL;
	p_bAWOpenIsHomed : REFERENCE TO BOOL;
	p_diAWOpenActualPos : REFERENCE TO DINT;
	p_bAWOpenFwdLmtSen : REFERENCE TO BOOL;
	p_bAWOpenRevLmtSen : REFERENCE TO BOOL;
	p_sAWOpenAxisErrTxt : REFERENCE TO STRING[80];
	p_bAWOpenJogging : REFERENCE TO BOOL;
	p_bAWOpenOpenSen : REFERENCE TO BOOL;
	p_bAWOpenCloseSen : REFERENCE TO BOOL;
END_VAR
(**)
VAR
	p_eInvertStat : REFERENCE TO eMotorBrkAction;
	p_eInvertStatus : REFERENCE TO eFBStatus;
	p_sInvertStatTxt : REFERENCE TO STRING[200];
END_VAR
(**)
VAR
	p_eOpsStat : REFERENCE TO eOperationsAction;
	p_eOpsStatus : REFERENCE TO eFBStatus;
	p_sOpsStatTxt : REFERENCE TO STRING[200];
	p_eOpsOpsStatus : REFERENCE TO eOperationsStatus;
	p_bOpsStatusRun : REFERENCE TO BOOL;
	p_bOpsStatusStop : REFERENCE TO BOOL;
	p_bOpsStatusCycleStop : REFERENCE TO BOOL;
	p_bOpsStatusStep : REFERENCE TO BOOL;
	p_bOpsUSStandby : REFERENCE TO BOOL;
	p_bOpsDSStandby : REFERENCE TO BOOL;
	p_bOpsRun : REFERENCE TO BOOL;
END_VAR
(**)
VAR
	p_sOpsInvertStepTxt : REFERENCE TO STRING[80];
	p_eOpsInvertCurrPos : REFERENCE TO eInvertPos;
END_VAR
(**)
VAR
	p_bOpsInvertStepInitConv : REFERENCE TO BOOL;
	p_bOpsInvertStepInitDone : REFERENCE TO BOOL;
END_VAR
(**)
VAR
	p_bOpsInvertStepAWMove : REFERENCE TO BOOL;
	p_bOpsSafeMode : REFERENCE TO BOOL;
END_VAR
(**)
VAR
	p_bOpsInvOnceTwicePCBOut : REFERENCE TO BOOL;
	p_bOpsInvertStepUSStandby : REFERENCE TO BOOL;
END_VAR
(**)
VAR
	p_eHermesStat : REFERENCE TO eHermesAction;
	p_eHermesStatus : REFERENCE TO eFBStatus;
	p_tyHermesConfiguration : REFERENCE TO tyHermesConfiguration;
END_VAR
(**)
VAR
	p_eLFLeaderStat : REFERENCE TO eLFAction;
	p_eLFLeaderStatus : REFERENCE TO eFBStatus;
	p_tyLFLeaderFollowerInfo : REFERENCE TO ARRAY[1..c_diLFClntNum] OF tyLFFollowerInfo;
	p_tyLFLeaderFollowerToLeaderTag : REFERENCE TO ARRAY[1..c_diLFClntNum] OF tyLFFollowerToLeaderTag;
END_VAR
(**)
VAR
	p_bLFFollowerProdAccDataMnl : REFERENCE TO BOOL;
	p_bLFFollowerLdrSeqCtrlInActive : REFERENCE TO BOOL;
	p_bLFFollowerUSAllow : REFERENCE TO BOOL;
	p_bLFFollowerDSAllow : REFERENCE TO BOOL;
END_VAR
(**)
VAR
	p_bFollower1WaitRlsProd : REFERENCE TO BOOL;
END_VAR
(**)
VAR
	p_bLCSLFAccDataMnl : REFERENCE TO BOOL;
END_VAR
(**)
VAR
	p_tyDI : REFERENCE TO tyDigitalInput;
END_VAR
(**)
VAR
	p_tyDO : REFERENCE TO tyDigitalOutput;
	p_eDOStat : REFERENCE TO eDOAction;
	p_eDOStatus : REFERENCE TO eFBStatus;
END_VAR
(**)
VAR
	p_eStopperStat : REFERENCE TO ePneuAction;
	p_eStopperStatus : REFERENCE TO eFBStatus;
	p_sStopperStatTxt : REFERENCE TO STRING[200];
	p_bStopperTwoCtrlOut : REFERENCE TO BOOL;
	p_bStopperExtCtrl : REFERENCE TO BOOL;
	p_bStopperRetCtrl : REFERENCE TO BOOL;
	p_bStopperExtended : REFERENCE TO BOOL;
END_VAR
(**)
VAR
	p_eClampStat : REFERENCE TO ePneuAction;
	p_eClampStatus : REFERENCE TO eFBStatus;
	p_sClampStatTxt : REFERENCE TO STRING[200];
	p_bClampTwoCtrlOut : REFERENCE TO BOOL;
	p_bClampExtCtrl : REFERENCE TO BOOL;
	p_bClampRetCtrl : REFERENCE TO BOOL;
END_VAR
(**)
VAR
	p_eInShutterStat : REFERENCE TO ePneuAction;
	p_eInShutterStatus : REFERENCE TO eFBStatus;
	p_sInShutterStatTxt : REFERENCE TO STRING[200];
	p_bInShutterExtCtrl : REFERENCE TO BOOL;
	p_bInShutterRetCtrl : REFERENCE TO BOOL;
	p_bInShutterTwoCtrlOut : REFERENCE TO BOOL;
	p_bInShutterExtended : REFERENCE TO BOOL;
	p_bInShutterRetracted : REFERENCE TO BOOL;
END_VAR
(**)
VAR
	p_eOutShutterStat : REFERENCE TO ePneuAction;
	p_eOutShutterStatus : REFERENCE TO eFBStatus;
	p_sOutShutterStatTxt : REFERENCE TO STRING[200];
	p_bOutShutterExtCtrl : REFERENCE TO BOOL;
	p_bOutShutterRetCtrl : REFERENCE TO BOOL;
	p_bOutShutterTwoCtrlOut : REFERENCE TO BOOL;
	p_bOutShutterExtended : REFERENCE TO BOOL;
	p_bOutShutterRetracted : REFERENCE TO BOOL;
END_VAR
(**)
VAR
	p_eClamp1Stat : REFERENCE TO ePneuAction;
	p_eClamp1Status : REFERENCE TO eFBStatus;
	p_sClamp1StatTxt : REFERENCE TO STRING[200];
	p_bClamp1ExtCtrl : REFERENCE TO BOOL;
	p_bClamp1RetCtrl : REFERENCE TO BOOL;
	p_bClamp1TwoCtrlOut : REFERENCE TO BOOL;
	p_bClamp1Extended : REFERENCE TO BOOL;
	p_bClamp1Retracted : REFERENCE TO BOOL;
END_VAR
(**)
VAR
	p_eClamp2Stat : REFERENCE TO ePneuAction;
	p_eClamp2Status : REFERENCE TO eFBStatus;
	p_sClamp2StatTxt : REFERENCE TO STRING[200];
	p_bClamp2ExtCtrl : REFERENCE TO BOOL;
	p_bClamp2RetCtrl : REFERENCE TO BOOL;
	p_bClamp2TwoCtrlOut : REFERENCE TO BOOL;
	p_bClamp2Extended : REFERENCE TO BOOL;
	p_bClamp2Retracted : REFERENCE TO BOOL;
END_VAR
(**)
VAR
	p_eClamp3Stat : REFERENCE TO ePneuAction;
	p_eClamp3Status : REFERENCE TO eFBStatus;
	p_sClamp3StatTxt : REFERENCE TO STRING[200];
	p_bClamp3ExtCtrl : REFERENCE TO BOOL;
	p_bClamp3RetCtrl : REFERENCE TO BOOL;
	p_bClamp3TwoCtrlOut : REFERENCE TO BOOL;
	p_bClamp3Extended : REFERENCE TO BOOL;
	p_bClamp3Retracted : REFERENCE TO BOOL;
END_VAR
(**)
VAR
	p_bMtrBrkRls : REFERENCE TO BOOL;
END_VAR
(*Insert your comment here.*)
VAR
	p_bLeftSen : REFERENCE TO BOOL;
	p_bRightSen : REFERENCE TO BOOL;
	p_diInitTm : REFERENCE TO DINT;
	p_eDirection : REFERENCE TO eConvDir;
END_VAR
(**)
VAR
	p_bConvAlmData : REFERENCE TO tyAlmDat;
	p_bDSSMEMAAlmData : REFERENCE TO tyAlmDat;
END_VAR
(**)
VAR
	p_bUnlockCovPrep : REFERENCE TO BOOL;
	p_bMachineSafetyPrep : REFERENCE TO BOOL;
END_VAR
(*Simulation*)
VAR
	p_eSimuStat : REFERENCE TO eSimulationsAction;
	p_eSimuStatus : REFERENCE TO eFBStatus;
	p_eSimuSimuStatus : REFERENCE TO eSimulationsStatus;
	p_bSimuStatusRun : REFERENCE TO BOOL;
	p_bSimuStatusStop : REFERENCE TO BOOL;
	p_bSimuStatusCycleStop : REFERENCE TO BOOL;
	p_bSimuStatusStep : REFERENCE TO BOOL;
END_VAR
(**)
VAR
	p_bUIBtnSectionLdr : REFERENCE TO BOOL;
	p_bLCSSectionLeaderEn : REFERENCE TO BOOL;
END_VAR
```

#### Local.var - Change By Project
```iecst
(*2020-10-08*)
(**)
(*Local Action & State & Status*)
VAR
	eAct : eUIAction := UIActIdle;
	eStat : eUIAction := UIActIdle;
	eStatus : eFBStatus := Idle;
	sStatTxt : STRING[200] := '';
	a_sStatText : ARRAY[0..50] OF STRING[200] := ['Idling','Initializing UI Page',49('')];
END_VAR
(**)
(*All General Alarm*)
VAR
	tyUIAlmData : tyUIAllAlm;
END_VAR
(**)
(*Local Output*)
VAR
	eStartupAct : eStartupAction;
	eHWInfoAct : eHWInfoAction;
	eTLBuzAct : eTLBuzAction;
	eRstErrAct : eRstErrAction;
	eProdRcpAct : eProdRcpAction;
	eMpProdRcpAct : eMpProdRcpAction;
	eMcParamAct : eMcParamAction;
	eUsrMgmtAct : eUsrMgmtAction;
	eUSSMEMAAct : eSMEMAAction;
	eDSSMEMAAct : eSMEMAAction;
	eUSSMEMA2Act : eSMEMAAction;
	eStopperAct : ePneuAction;
	eConvAct : eConvAction;
	eAWOpenAct : eAWAction;
	eInvertAct : eMotorBrkAction;
	eOpsAct : eOperationsAction;
	eHermesAct : eHermesAction;
	eLFLeaderAct : eLFAction;
	eDOAct : eDOAction;
	eClampAct : ePneuAction;
	eInShutterAct : ePneuAction;
	eOutShutterAct : ePneuAction;
	eClamp1Act : ePneuAction;
	eClamp2Act : ePneuAction;
	eClamp3Act : ePneuAction;
	eSimuAct : eSimulationsAction;
END_VAR
(**)
VAR
	tyMcParamWr : tyMcParam;
	tyProdRcpInfoIn : tyProdRcpParam;
	tyProdRcpCurrRcpWr : tyProdRcpParam;
	sProdRcpSearch : STRING[30];
	sProdRcpScan : STRING[30];
	tyUsrMgmtInfoIn : tyUsrMgmtParam;
	tyUsrMgmtAccessRightLvl1Wr : tyUsrMgmtAccessRight;
	tyUsrMgmtAccessRightLvl2Wr : tyUsrMgmtAccessRight;
	tyUsrMgmtAccessRightLvl3Wr : tyUsrMgmtAccessRight;
	a_tyHermesUSParamWr : ARRAY[0..c_diHermesConfigMaxIdx] OF tyHermesUSParam;
	a_tyHermesDSParamWr : ARRAY[0..c_diHermesConfigMaxIdx] OF tyHermesDSParam;
	tyHermesSvyParamWr : tyHermesSvyParam;
	sSetIPAddr : STRING[15];
	sSetSubnetMask : STRING[15];
	bManualMod : BOOL;
	bUIManualMod : BOOL;
	bMuteBuz : BOOL;
	diMnlAWGoWidth : DINT;
	diMnlAWNomSpd : DINT;
	diMnlAWTargetPos : DINT;
	diMnlAWStepSize : DINT;
	diMnlAWJogSpd : DINT;
	diMnlInvertNomSpd : DINT;
	diMnlInvertTargetPos : DINT;
	diMnlInvertStepSize : DINT;
	diMnlInvertJogSpd : DINT;
	bVSMEMAUSEn : BOOL;
	bVSMEMADSEn : BOOL;
	bVSMEMAUBA : BOOL;
	bVSMEMAUBAStat : BOOL;
	bVSMEMADSB : BOOL;
	bVSMEMAUS2En : BOOL;
	bVSMEMAUBA2 : BOOL;
	bVSMEMAUBAStat2 : BOOL;
	bLeaderRun : BOOL;
	bProdAccData : BOOL;
	bOpsBypsInitConv : BOOL;
	bRlsNewProd : BOOL;
	bCheckDone : BOOL;
	bFilterSortP0400 : BOOL;
	bFilterSortP1040 : BOOL;
	bUpdateP0400Table : BOOL;
	bUpdateP1040Table : BOOL;
	bMnlModMachineSafetySigToDS : BOOL;
	bMnlModUnlockCover1Req : BOOL;
	bMnlModCoverPBLED1 : BOOL;
	bMnlModBypassTopCover1 : BOOL;
	bMnlModTopCoverSwitch1 : BOOL;
	bRtnBrdReset : BOOL;
	bSimuMod : BOOL;
END_VAR
(**)
(*Local Input*)
(**)
(*Local*)
VAR
	bInitDone : BOOL;
	bInitialDone : BOOL;
	i : UINT := 0;
	eUIInit : eUIInitial := UIInitialC0005;
	usiChgPage : USINT := 1;
	eCurrPage : ePage := UIP0001Startup;
	eChgPage : ePage := UIP0001Startup;
	eChgPageOld : ePage := UIP0001Startup;
	bChgPage : BOOL := FALSE;
	bLoginSuccess : BOOL := FALSE;
	bJogFast : BOOL := FALSE;
	bJogSlow : BOOL := FALSE;
	bJogStopAW : BOOL := FALSE;
	bOnlineTemp : BOOL := FALSE;
	bIPDuplicate : BOOL := FALSE;
	bRefreshProdRcpDetail : BOOL := FALSE;
	bRefreshProdRcpTable : BOOL := TRUE;
	bRefreshUsrMgmtTable : BOOL := TRUE;
	bTeachStopperAtLftPos : BOOL := FALSE;
	bTeachStopperAtRgtPos : BOOL := FALSE;
	usiConvStep : USINT := 0;
	usiLoginStep : USINT := 0;
	usiSelProdRcpStep : USINT := 0;
	usiSaveProdRcpStep : USINT := 0;
	usiDelProdRcpStep : USINT := 0;
	usiProdRcpToXMLStep : USINT := 0;
	usiProdRcpFromXMLStep : USINT := 0;
	usiEditUsrMgmtStep : USINT := 0;
	usiSaveUsrMgmtStep : USINT := 0;
	usiDelUsrMgmtStep : USINT := 0;
	usiSaveCommStep : USINT := 0;
	usiSaveIPAddrStep : USINT := 0;
	usiSaveSubnetMaskStep : USINT := 0;
	usiDelMcDetailsStep : USINT := 0;
	usiTableShftStep : USINT := 0;
	usiLFLeaderCtrlStep : USINT := 0;
	uiSSaverCnt : UINT := 0;
	fbSSaverTm : TON;
	fbErrBlinkTm : TON := (IN:=FALSE,PT:=T#1s,Q:=FALSE,ET:=0,StartTime:=0,M:=FALSE,Restart:=0);
	fbRstBlinkTm : TON := (IN:=FALSE,PT:=T#1s,Q:=FALSE,ET:=0,StartTime:=0,M:=FALSE,Restart:=0);
	fbStopBlinkTm : TON := (IN:=FALSE,PT:=T#500ms,Q:=FALSE,ET:=0,StartTime:=0,M:=FALSE,Restart:=0);
	fbMcStatUpdtTm : TON := (IN:=FALSE,PT:=T#0.5s,Q:=FALSE,ET:=0,StartTime:=0,M:=FALSE);
	fbAccDatBlinkTm : TON := (IN:=FALSE,PT:=T#500ms,Q:=FALSE,ET:=0,StartTime:=0,M:=FALSE,Restart:=0);
	fbRlsNewProdBlinkTm : TON := (IN:=FALSE,PT:=T#500ms,Q:=FALSE,ET:=0,StartTime:=0,M:=FALSE,Restart:=0);
	fbBypsInitConvBlinkTm : TON := (IN:=FALSE,PT:=T#500ms,Q:=FALSE,ET:=0,StartTime:=0,M:=FALSE,Restart:=0);
	fbLFLeaderCtrlBlinkTm : TON := (IN:=FALSE,PT:=T#500ms,Q:=FALSE,ET:=0,StartTime:=0,M:=FALSE,Restart:=0);
	fbLmtRstTm : TON := (PT:=T#1s);
	fbJogSlowToFastDlyTm : TON := (IN:=FALSE,PT:=T#2s,Q:=FALSE,ET:=0,StartTime:=0,M:=FALSE,Restart:=0);
	fbLoadingWarmUpTm : TON := (IN:=FALSE,PT:=T#5s,Q:=FALSE,ET:=0,StartTime:=0,M:=FALSE,Restart:=0);
	fbLoadingLogoTm : TON := (IN:=FALSE,PT:=T#151ms,Q:=FALSE,ET:=0,StartTime:=0,M:=FALSE,Restart:=0);
	tyP0400Table : tyTable := (bSliderActive:=FALSE,bTableActive:=FALSE,sVisuNm:='Visu',uiSelectedRow:=1,uiSelectedRowOld:=1,uiTablePos:=1);
	fbP0400Table : fbTableCtrl;
	tyP0700Table : tyTable := (bSliderActive:=FALSE,bTableActive:=FALSE,sVisuNm:='Visu',uiSelectedRow:=1,uiSelectedRowOld:=1,uiTablePos:=1);
	fbP0700Table : fbTableCtrl;
	tyP1040Table : tyTable := (bSliderActive:=FALSE,bTableActive:=FALSE,sVisuNm:='Visu',uiSelectedRow:=1,uiSelectedRowOld:=1,uiTablePos:=1);
	fbP1040Table : fbTableCtrl_v2;
	tyP1050Table : tyTable := (bSliderActive:=FALSE,bTableActive:=FALSE,sVisuNm:='Visu',uiSelectedRow:=1,uiSelectedRowOld:=1,uiTablePos:=1);
	fbP1050Table : fbTableCtrl;
	tyP1080Table : tyTable := (bSliderActive:=FALSE,bTableActive:=FALSE,sVisuNm:='Visu');
	fbP1080Table : fbTableCtrl;
	udiP1040SelectedRow : UDINT := 0;
	udiP1040SelectedRowOld : UDINT := 0;
	usiP1080SelectedLvl : USINT := 0;
	udiP1080SelectedRow : UDINT := 0;
	a_iIPPart1 : ARRAY[1..4] OF INT := [4(0)];
	a_iIPPart2 : ARRAY[1..4] OF INT := [4(0)];
	a_iSubnetMaskPart1 : ARRAY[1..4] OF INT := [4(0)];
	sLFIPAddrTemp : STRING[15];
	sElapseTm : STRING[80] := '';
	udiElapseTm : UDINT := 0;
END_VAR
(**)
(*Local*)
VAR
	bDSTranErr : BOOL;
	bChgPageDone : BOOL;
	bPromptSessionExp : BOOL := FALSE;
	fbAutoLogoutTm : TON;
	fbTouchTm : fbTouchGetAction := (sVisuNm:='Visu');
	bUpdateP1040LoadData : BOOL;
	bLFRunInBG : BOOL;
	bLFDeleteOn : BOOL;
	bUpdateP1050Table : BOOL;
	iIPExtract : INT;
	sLFSettingCurrentIP : STRING[4];
	iLFSettingCurrentIP : INT;
	sLFSettingAutoFill : STRING[15];
	sLFSettingTemp : STRING[15];
	bLFSettingAutoFill : BOOL;
	bLFSettingAutoClear : BOOL;
END_VAR
(**)
VAR
	bLoadingScreen : BOOL;
END_VAR
(**)
VAR
	sTempIPAddr : STRING[15];
	sTempSubnetMask : STRING[15];
	udiTempEthMode : UDINT;
	bTempAddrFillDone : BOOL;
	bUpdateP1021Network : BOOL;
	bMismatchOverWriteConfig : BOOL;
	bIPConfigChgDone : BOOL;
	bOverwriteIP : BOOL;
	bOverwriteSubnet : BOOL;
	bOverwriteEthMode : BOOL;
	usiNetworkModeOld : USINT;
	usiNetworkModeNew : USINT;
	usiNetworkModeSelected : USINT;
	usiChgNetworkConfigStep : USINT := 0;
	usiRefreshDetailStep : USINT := 0;
	bSaveNetworkPriority : BOOL;
	bNetworkConfigChanged : BOOL;
	uiLFStartEditNo : UINT;
END_VAR
(**)
VAR
	uiSongIndex : UINT;
	bSongEn : BOOL;
END_VAR
(**)
VAR
	bCoverPB1Timer : BOOL := FALSE;
	bCoverPBLED1 : BOOL;
	fbCoverPB1CountDownTm : TON := (IN:=FALSE,PT:=T#5s,Q:=FALSE,ET:=0,StartTime:=0,M:=FALSE,Restart:=0);
	fbCoverPBLED1BlinkTm : TON := (IN:=FALSE,PT:=T#200ms,Q:=FALSE,ET:=0,StartTime:=0,M:=FALSE,Restart:=0);
	bBypassTopCover1 : BOOL;
	bBypassTopCoverPB1 : BOOL;
	bMachineSafetySigToUS : BOOL;
	bMachineSafetySigToDS : BOOL;
	bTopCoverSwitchCoil1 : BOOL;
	bBypsTopCover : BOOL;
	bUnlockCover1Req : BOOL;
END_VAR
(*Hermes 1.3*)
VAR
	bSaveHMISvyConfig : BOOL;
	bSaveHMIConfigure : BOOL;
	bQueryBoardInfo : BOOL;
	bNaviLyr1 : BOOL;
	bNaviLyr2 : BOOL;
END_VAR
```

#### Local.typ - Change By Project
```iecst
(*2020-10-08*)
(**)

TYPE
	ePage :
		(
		UIP0000SSaver := 0, (*Page Screen Saver*)
		UIP0001Startup := 1, (*Page Startup*)
		UIP0002Menu := 2, (*Page Menu*)
		UIP0100Login := 100, (*Page Login*)
		UIP0200OpsGen := 200, (*Page Operation*)
		UIP0201OpsConv := 201, (*Page Operation*)
		UIP0300McInfo := 300, (*Page Machine Info*)
		UIP0400ProdSel := 400, (*Page Product Selection*)
		UIP0600Alm := 600, (*Page Alarm*)
		UIP0700LFCtrl := 700, (*Page Leader Follower Control*)
		UIP0900GenIn := 900, (*Page General Input*)
		UIP0910GenOut := 910, (*Page General Output*)
		UIP0920MtrNPneuCtrl := 920, (*Page Motor And Pneumatic Control*)
		UIP0921ClampNoRS := 921, (*Page Stopper*)
		UIP0922Shutter := 922, (*Page Shutter*)
		UIP0923Stopper := 923, (*Page Stopper*)
		UIP0924ClampWithRS := 924, (*Page Stopper*)
		UIP0931ConvInv := 931, (*Page Conveyor*)
		UIP0934AW := 934, (*Page Auto Width*)
		UIP0940CommCtrl := 940, (*Page Communication Control*)
		UIP0950Simu := 950, (*Page Simu*)
		UIP1000Lang := 1000, (*Page Language And Setup*)
		UIP1020McSetNavi := 1020, (*Page Machine Setting - Navigation*)
		UIP1021McSetGen := 1021, (*Page Machine Setting - General*)
		UIP1022McSetVComm := 1022, (*Page Machine Setting - Vertical Communication*)
		UIP1023McSetHComm := 1023, (*Page Machine Setting - Horizontal Communication*)
		UIP1024McSetAntiGap := 1024, (*Page Machine Setting - Anti-Gap*)
		UIP1040ProdSet := 1040, (*Page Product Setting*)
		UIP1050LFSet := 1050, (*Page Leader Follower Setting*)
		UIP1080UsrMgmt := 1080, (*Page User Management*)
		UIP1081UsrMgmtUsrAccessRgt := 1081 (*Page User Management - Access Right*)
		);
	tyTable : 	STRUCT
		bSliderActive : BOOL := FALSE;
		bTableActive : BOOL := FALSE;
		sVisuNm : STRING[80] := 'Visu';
		uiSelectedRow : UINT := 1;
		uiSelectedRowOld : UINT := 1;
		uiTablePos : UINT := 1;
	END_STRUCT;
END_TYPE
```
